# EPICS autosave request: iocBoot/iocTomoScan_prisma/auto_settings.req
file "tomoScan_settings.req", P=$(P), R=$(R)
#file "tomoScan_PSO_settings.req", P=$(P), R=$(R)
file "tomoScan_prisma_settings.req", P=$(P), R=$(R)
